FUNCTION_BLOCK FB_ElementIterator IMPLEMENTS I_ElementIterator
VAR_INPUT
END_VAR
VAR_OUTPUT
END_VAR
VAR
	_pElementData		: POINTER TO ST_Element;
	_diNumOfElements	: DINT;
	_diIndex			: DINT;
END_VAR

METHOD hasNext : BOOL
VAR
	
END_VAR
IF _pElementData = 0 THEN
	RETURN;
END_IF

hasNext := _diIndex < _diNumOfElements;
END_METHOD

METHOD init : BOOL
VAR_IN_OUT
	io_astElements	:ARRAY[*] OF ST_Element;
END_VAR
_pElementData 		:= io_astElements;
_diNumOfElements 	:= UPPER_BOUND(io_astElements, 1);
_diIndex			:= LOWER_BOUND(io_astElements, 1);
END_METHOD

METHOD next : ST_Element
VAR
	stElement :ST_Element;
END_VAR
IF _pElementData = 0 THEN
	RETURN;
END_IF

IF _diIndex < _diNumOfElements THEN
	MEMCPY(srcAddr:= (_pElementData + (_diIndex * SIZEOF(stElement))), destAddr:= ADR(stElement), n:= SIZEOF(stElement));
	next := stElement;
	_diIndex := _diIndex + 1;
END_IF
END_METHOD

END_FUNCTION_BLOCK

(* stored: Version 1.1.0.1
   POU FB_ElementIterator: Id {286cbf6e-9d81-4be3-b012-a4a90e1fb91e}, SpecialFunc None
   Method hasNext: Id {e35d0595-4a25-4de0-9938-125e4881d2a7}
   Method init: Id {b63e8828-6048-4c9a-95fb-f76d10f8c2b8}
   Method next: Id {b0abfcdf-40eb-4e50-90de-678e65291584} *)
